{attribute 'linkalways'} 
{attribute 'no_explicit_call' := 'This FB is a CLASS and must be accessed using methods or properties'}
{attribute 'enable_dynamic_creation'}
FUNCTION_BLOCK _TcVnVector2_DINT EXTENDS AliasDatatypeBase
VAR
	localData : TcVnVector2_DINT;
	activeData : REFERENCE TO TcVnVector2_DINT REF= localData;
	aliasBaseDatatype : _Array0to1OfDINT;
END_VAR

PROPERTY PUBLIC Address : PVOID
GET
Address := ADR(activeData);
END_GET
END_PROPERTY

METHOD PUBLIC ClearReference
VAR_INPUT
END_VAR
activeData REF= localData;
SetBaseDatatypeReference();
END_METHOD

METHOD PUBLIC Clone : I_Datatype
VAR
    pClone : POINTER TO _TcVnVector2_DINT;
END_VAR
pClone := __NEW(_TcVnVector2_DINT);
Clone := pClone^;
END_METHOD

METHOD FB_init : BOOL
VAR_INPUT
	bInitRetains : BOOL; // if TRUE, the retain variables are initialized (warm start / cold start)
	bInCopyCode : BOOL;  // if TRUE, the instance afterwards gets moved into the copy code (online change)
	//InitialValue : <type>; // if possible, not all values can be initialized
END_VAR
//localData := InitialValue; // if possible, not all values can be initialized
SetBaseDatatypeReference();
AddBaseDatatype(aliasBaseDatatype);
END_METHOD

PROPERTY PUBLIC Identifier : T_MAXSTRING
GET
Identifier := 'TcVnVector2_DINT';
END_GET
END_PROPERTY

METHOD PUBLIC MakeReferenceTo
VAR_INPUT
	ReferenceTarget : REFERENCE TO TcVnVector2_DINT;
END_VAR
activeData REF= ReferenceTarget;
SetBaseDatatypeReference();
END_METHOD

METHOD PROTECTED SetBaseDatatypeReference
VAR_INPUT
END_VAR
aliasBaseDatatype.MakeReferenceTo(activeData);
END_METHOD

PROPERTY PUBLIC Size : UDINT
GET
Size := SIZEOF(activeData);
END_GET
END_PROPERTY

METHOD TryMakeReferenceTo : BOOL
VAR_INPUT
	Target : I_Datatype;
END_VAR
VAR
	targetAsAlias : I_AliasDatatype;
	pTargetData : POINTER TO TcVnVector2_DINT;
END_VAR
IF NOT Target.TryResolveAsAliasDatatype(targetAsAlias) THEN
	RETURN;
END_IF

IF targetAsAlias.Identifier <> Identifier THEN
	RETURN;
END_IF

pTargetData := Target.Address;
activeData REF= pTargetData^;
SetBaseDatatypeReference();
TryMakeReferenceTo := TRUE;
END_METHOD

PROPERTY PUBLIC Value : REFERENCE TO TcVnVector2_DINT
GET
Value REF= activeData;
END_GET
END_PROPERTY

END_FUNCTION_BLOCK

(* stored: Version 1.1.0.1, ProductVersion 3.1.4024.13
   POU _TcVnVector2_DINT: Id {30530a71-1a5e-0582-392c-8a8d4a83820f}, SpecialFunc None
   Folder Core: Id {f44bdcc0-718d-0b69-140d-cf9fea4ee0f6}
   Folder Protected: Id {238a52d6-6497-0087-3864-3ce0c5b4c78b}
   Folder Customize: Id {b1219068-8501-0eab-319b-b45e8c6fbb06}
   Folder Constructor: Id {dd789b49-f5c2-0eeb-173c-cfb588c57e31}
   Property Address: Id {ada31421-8531-031e-293e-1b1d47c5f1e7}
   Get Get: Id {66ce5751-80c9-04fe-3df3-c5382f984bb0}
   Method ClearReference: Id {58e2f381-6329-0744-3a78-dfbd11edf129}
   Method Clone: Id {e0ae9401-9afe-0b63-3bbd-d6547c518553}
   Method FB_init: Id {e102e272-c09b-0476-21e5-23887278e033}
   Property Identifier: Id {c6d58249-ade7-089f-2201-be1a98d58cac}
   Get Get: Id {6577af0e-2b03-02f1-18f6-c8618558fb9b}
   Method MakeReferenceTo: Id {5587e013-a4b4-05e5-19af-7c817dd8fb8a}
   Method SetBaseDatatypeReference: Id {f154c024-a59d-06e9-3e5d-acb230e12018}
   Property Size: Id {85298c3a-b9a1-0f9e-2c62-6a586a3d5743}
   Get Get: Id {66074d22-4026-098f-16bc-fd37a9e67e30}
   Method TryMakeReferenceTo: Id {58478c9e-a154-0eb3-31f9-3841fad6e99b}
   Property Value: Id {1eb39456-e949-0dcd-1e0a-f10ff6b8e13e}
   Get Get: Id {3eaa881e-34cc-09b8-3d4c-055cfa7701fb} *)
